FUNCTION_BLOCK FB_Stirrer
VAR_INPUT
	enable					:BOOL;
	continueTime			:LREAL;//Min   持续时间
	intervalTime			:LREAL;//Min  间隔时间
END_VAR
VAR_OUTPUT
	PumpWorkingF			:BOOL;//正转
	PumpWorkingB			:BOOL;//反转

END_VAR
VAR 
	ton_C:TON;	//   持续时间
	ton_I:TON;	//   持续时间
	step:INT;
	R_trig:R_TRIG;
	F_trig:F_TRIG;
	
END_VAR

R_trig(CLK:=enable , Q=> );
F_trig(CLK:=enable , Q=> );


IF F_trig.Q THEN 
	step:=0;
END_IF

CASE step OF
0://启动
	PumpWorkingF:=FALSE;
	PumpWorkingB:=FALSE;
	ton_C(IN:=FALSE);
	ton_I(IN:=FALSE);
	IF R_trig.Q THEN
	 	step:=10;		
	END_IF	
10://正转
	PumpWorkingF:=TRUE;
	PumpWorkingB:=FALSE;
	ton_I(IN:=FALSE);
	ton_C(IN:=TRUE  , PT:=LREAL_TO_TIME(continueTime*1000*60) , Q=> , ET=> );
	IF ton_C.Q THEN 		
		step:=20;
	END_IF	
20://间隔
	PumpWorkingF:=FALSE;
	PumpWorkingB:=FALSE;
	ton_C(IN:=FALSE);
	ton_I(IN:=TRUE , PT:=LREAL_TO_TIME(intervalTime*1000*60) , Q=> , ET=> );
	IF ton_I.Q THEN 
		step:=30;
	END_IF
30://反转
	PumpWorkingF:=FALSE;
	PumpWorkingB:=TRUE;
	ton_I(IN:=FALSE);
	ton_C(IN:=TRUE  , PT:=LREAL_TO_TIME(continueTime*1000*60) , Q=> , ET=> );
	IF ton_C.Q THEN 		
		step:=40;
	END_IF	
40://间隔
	PumpWorkingF:=FALSE;
	PumpWorkingB:=FALSE;
	ton_C(IN:=FALSE);
	ton_I(IN:=TRUE , PT:=LREAL_TO_TIME(intervalTime*1000*60) , Q=> , ET=> );
	IF ton_I.Q THEN 
		step:=10;
	END_IF

END_CASE

END_FUNCTION_BLOCK

(* stored: Version 1.1.0.1, ProductVersion 3.1.4024.11
   POU FB_Stirrer: Id {e53c1647-df9f-4491-92a0-6b57a015c043}, SpecialFunc None *)
